Staubli VAL3: getBitAt.pgx

public program getBitAt(num x_nByteIndex, num x_nBitIndex, num& x_nBuffer[], bool& x_bRes)
  local string l_sMask
  local string l_sByte
  local string l_sResult
  local num l_nResult
begin

  if x_nBitIndex>7
    x_bRes=false
    return
  endIf

  call bitOp:DecToBin(x_nBuffer[x_nByteIndex], l_sByte)
  call bitOp:DecToBin(power(2, x_nBitIndex), l_sMask)
  call bitOp:boolAnd(l_sByte, l_sMask, l_sResult)

  call bitOp:BinToDec(l_sResult, l_nResult)
  if l_nResult>0
    x_bRes=true
  else
    x_bRes=false
  endIf

end
